DATA_BLOCK "R_TRIG_DB"
AUTHOR : SIMATIC
FAMILY : BIT
NAME : R_TRIG
VERSION : 1.0
NON_RETAIN
R_TRIG

BEGIN

END_DATA_BLOCK

